VAR_GLOBAL CONSTANT
	SS_INITIALIZE: SINT := 0;
	SS_STEP: SINT := 1;
END_VAR

(* stored: Version 1.1.0.1, ProductVersion 3.1.4024.10
   GVL CodeGeneration: Id {83550502-77a3-4a1e-98c2-7fa46eeae05b} *)
